(* Logix 5000 project; controller Week_4_PLC_1_Compute_CPT Emulate 5570 rev 30.12; software revision 30.01 *)

TASK MainTask (continuous, watchdog 500 ms) : MainProgram

MODULES
   Local : Emulate 5570 (ICP 2, rev 30.12)
END_MODULES

PROGRAM MainProgram   (* main routine MainRoutine *)
VAR
   Counter1 : COUNTER := (PRE := 10);
   Counter2 : COUNTER := (PRE := 5);
   PB1 : BOOL;
   Value1 : DINT;
END_VAR

ROUTINE MainRoutine   (* ladder *)
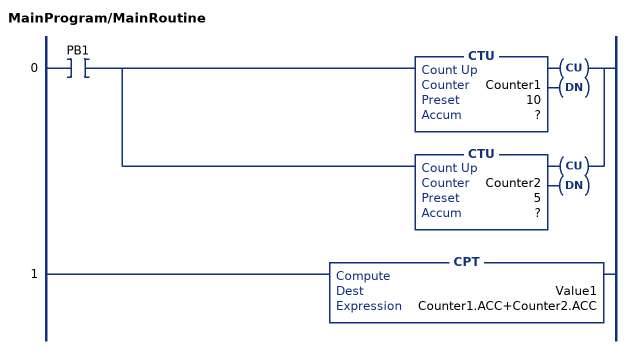
   0: XIC(PB1)[CTU(Counter1,?,?) ,CTU(Counter2,?,?) ];
   1: CPT(Value1,Counter1.ACC+Counter2.ACC);
END_ROUTINE
END_PROGRAM
